// TIA Portal project "filling tankk" (V16)
// Vorlageprojekt für das Buch mit Zielsystem S7-1200

(* hardware
DEVICE "S7-1200-Station_1"  S7-1200 Station
   slot 0: "Baugruppenträger_0"  Rack  V1.0
   slot 1: "PLC_1"  CPU 1211C DC/DC/DC  6ES7 211-1AE40-0XB0  V4.1
*)

// ===== PLC "PLC_1"  CPU 1211C DC/DC/DC =====

VAR_GLOBAL   // PLC tag table "Standard-Variablentabelle"
   "Tag_1" AT %A0.0 : Bool;
   "Tag_2" AT %E0.0 : Bool;
   "Tag_3" AT %E0.1 : Bool;
   "Tag_4" AT %I10.0 : Bool;
   "Tag_5" AT %Q10.0 : Bool;
   "Tag_6" AT %I10.1 : Bool;
   "Tag_7" AT %M0.0 : Bool;
   "Tag_8" AT %Q0.1 : Bool;
   "Tag_9" AT %M0.1 : Bool;
   "Tag_10" AT %M0.2 : Bool;
   "Tag_11" AT %M1.0 : Bool;
   "Tag_12" AT %M1.2 : Bool;
   "Tag_13" AT %M1.3 : Bool;
   "Tag_14" AT %Q0.2 : Bool;
END_VAR

// folder: System blocks/Program resources

DATA_BLOCK "t1"   // DB1
{ S7_Optimized_Access := 'TRUE' }
AUTHOR : Simatic
FAMILY : IEC
NAME : IEC_TMR
VERSION : 1.0
// stored: InstanceOfName IEC_TIMER
"IEC_TIMER"
BEGIN
END_DATA_BLOCK

DATA_BLOCK "t2"   // DB2
{ S7_Optimized_Access := 'TRUE' }
AUTHOR : Simatic
FAMILY : IEC
NAME : IEC_TMR
VERSION : 1.0
// stored: InstanceOfName IEC_TIMER
"IEC_TIMER"
BEGIN
END_DATA_BLOCK

// folder: (top level)

FUNCTION "MHJ-PLC-Lab-Function-S71200" : Void   // FC9000, SCL
{ S7_Optimized_Access := 'TRUE' }
VERSION : 0.1
   VAR_TEMP
      rdTimeReturn : Int;
      outputTime : DTL;
      SyncVal : Byte;
      forVal : Int;
      forVal_2 : Int;
      Value : Byte;
   END_VAR
   VAR CONSTANT
      CompVal : Byte := 16#34;
      Value_01 : Byte := 16#11;
      Value_01_DW : DWord := 16#A165_D992;
      Value_02_DW : DWord := 16#58BE_4401;
   END_VAR
BEGIN

   #Value:=PEEK(area := 16#82,
        dbNumber := 0,
        byteOffset := 511);
   #Value := #Value + 1;

   POKE(area := 16#82,
        dbNumber := 0,
        byteOffset := 511,
        value := #Value);

   POKE(area:=16#81,
        dbNumber:=0,
        byteOffset:=1016,
        value:=#Value_01_DW);
   POKE(area := 16#81,
        dbNumber := 0,
        byteOffset := 1020,
        value := #Value_02_DW);

   POKE(area := 16#81,
        dbNumber := 0,
        byteOffset := 511,
        value := B#16#00);

   FOR #forVal := 0 TO 120 DO
       FOR #forVal_2:=0 TO 10 DO
           #rdTimeReturn:=RD_SYS_T(#outputTime);
           #rdTimeReturn := WR_SYS_T(#outputTime);
           #rdTimeReturn := RD_SYS_T(#outputTime);
           #rdTimeReturn := WR_SYS_T(#outputTime);
       END_FOR;
       #SyncVal:= PEEK(area := 16#81,
                      dbNumber := 0,
                      byteOffset := 511);
       IF #SyncVal = #CompVal THEN
          GOTO M_1;
       END_IF;
   END_FOR;
   RETURN;

   M_1:
   POKE(area := 16#81,
        dbNumber := 0,
        byteOffset := 511,
        value := B#16#0);
END_FUNCTION

ORGANIZATION_BLOCK "Main"   // OB1, LAD, ProgramCycle
TITLE = "Main Program Sweep (Cycle)"
{ S7_Optimized_Access := 'TRUE' }
VERSION : 0.1
   VAR_INPUT
      Initial_Call : Bool;   // Initial call of this OB
      Remanence : Bool;   // =True, if remanent data are available
   END_VAR
BEGIN

REGION Network 1: Konnektierungsbaustein für PLC-Lab
   // Im Netzwerk 1 wird der Konnektierungsbaustein für PLC-Lab aufgerufen.
   // Dieser Aufruf darf nicht entfernt werden!
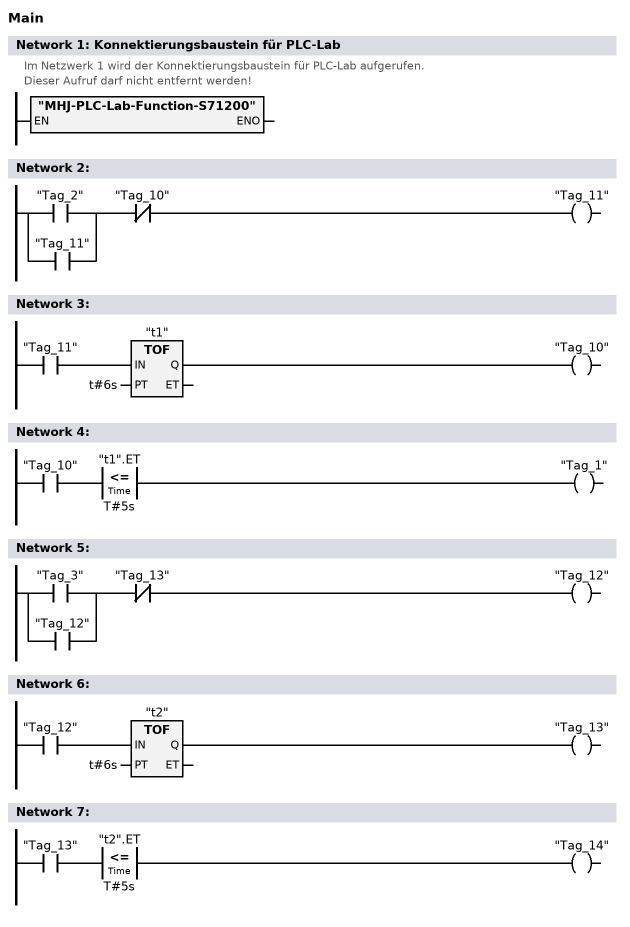
   RUNG wire#powerrail
      "MHJ-PLC-Lab-Function-S71200"()
   END_RUNG
   // the same network as SCL:
   "MHJ-PLC-Lab-Function-S71200"();
END_REGION

REGION Network 2
   RUNG wire#powerrail
      Contact( "Tag_2" )
      wire#w1
      I_Contact( "Tag_10" )
      Coil( "Tag_11" )
   END_RUNG
   RUNG wire#powerrail
      Contact( "Tag_11" )
   END_RUNG wire#w1
   // the same network as SCL:
   "Tag_11" := ("Tag_2" OR "Tag_11") AND NOT "Tag_10";
END_REGION

REGION Network 3
   "t1".TOF(IN := "Tag_11", PT := t#6s);
   "Tag_10" := "t1".Q;
END_REGION

REGION Network 4
   RUNG wire#powerrail
      Contact( "Tag_10" )
      { S7_Templates := "SrcType := Time" } LE_Contact(in1 := "t1".ET, in2 := T#5s)
      Coil( "Tag_1" )
   END_RUNG
   // the same network as SCL:
   "Tag_1" := "Tag_10" AND ("t1".ET <= T#5s);
END_REGION

REGION Network 5
   RUNG wire#powerrail
      Contact( "Tag_3" )
      wire#w1
      I_Contact( "Tag_13" )
      Coil( "Tag_12" )
   END_RUNG
   RUNG wire#powerrail
      Contact( "Tag_12" )
   END_RUNG wire#w1
   // the same network as SCL:
   "Tag_12" := ("Tag_3" OR "Tag_12") AND NOT "Tag_13";
END_REGION

REGION Network 6
   "t2".TOF(IN := "Tag_12", PT := t#6s);
   "Tag_13" := "t2".Q;
END_REGION

REGION Network 7
   RUNG wire#powerrail
      Contact( "Tag_13" )
      { S7_Templates := "SrcType := Time" } LE_Contact(in1 := "t2".ET, in2 := T#5s)
      Coil( "Tag_14" )
   END_RUNG
   // the same network as SCL:
   "Tag_14" := "Tag_13" AND ("t2".ET <= T#5s);
END_REGION
END_ORGANIZATION_BLOCK